TYPE ACRMemoryUIntEvents :
STRUCT
	_Values : ARRAY [0..GCL.cMemoryEventsMAX] OF ACRMemoryUIntEvent;
END_STRUCT
END_TYPE

(* stored: Version 1.1.0.1, ProductVersion 3.1.4020.12
   DUT ACRMemoryUIntEvents: Id {162ff785-5406-485c-9a8a-b0e0f1f9a37c} *)
